INTERFACE Istate

PROPERTY Description : STRING
GET
END_GET
END_PROPERTY

METHOD execute : BOOL
END_METHOD

END_INTERFACE

(* stored: Version 1.1.0.1
   Itf Istate: Id {cf3b1d54-4f51-4e95-8f09-e0bf534e3e62}
   Property Description: Id {f59e69a3-df26-4a9a-8375-62c52f4fd08c}
   Get Get: Id {c5175e1d-2229-4db5-9bca-cfca76f8cdc2}
   Method execute: Id {2b3674e8-71bd-45f9-8d83-3a8fcc14aa13} *)
